PROGRAM SerialCom
VAR
	fbSerialControl : SerialLineControlADS;
	fbSendString	: SendString;
	fbReceiveString	: ReceiveString;
	
	bBarcodeReceivedReset_FE: F_TRIG;
END_VAR

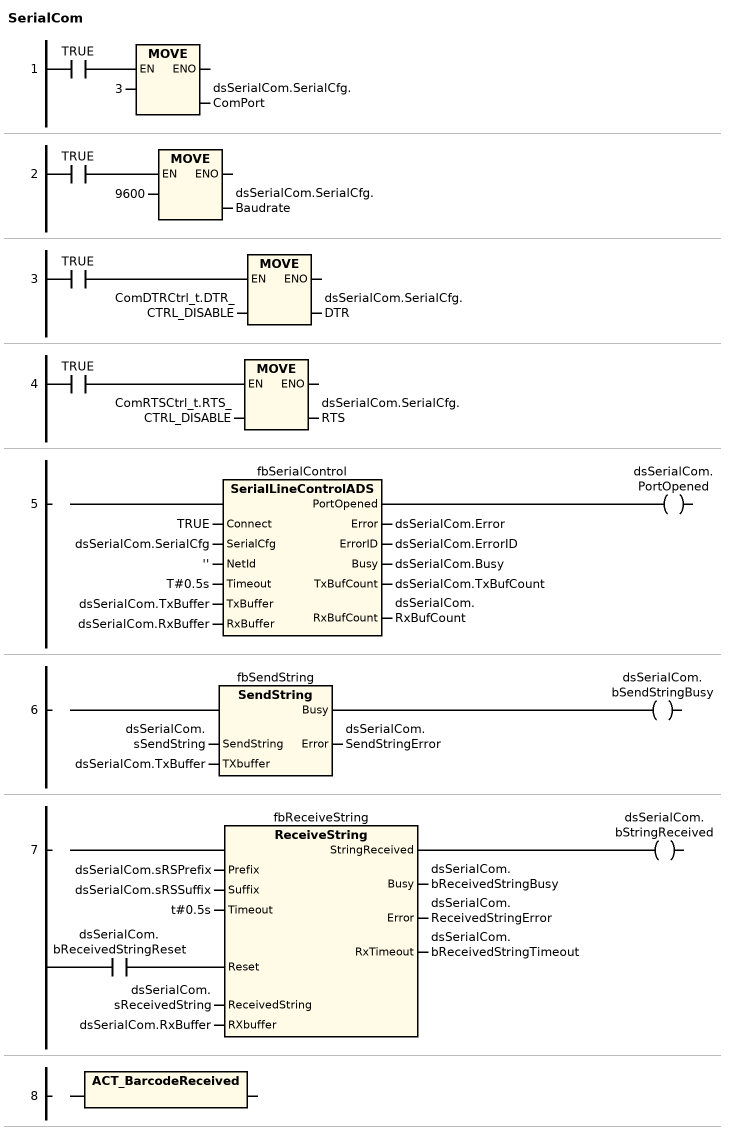
// NETWORK 1
dsSerialCom.SerialCfg.ComPort := 3;

// NETWORK 2
dsSerialCom.SerialCfg.Baudrate := 9600;

// NETWORK 3
dsSerialCom.SerialCfg.DTR := ComDTRCtrl_t.DTR_CTRL_DISABLE;

// NETWORK 4
dsSerialCom.SerialCfg.RTS := ComRTSCtrl_t.RTS_CTRL_DISABLE;

// NETWORK 5
fbSerialControl(
    Connect := TRUE,
    SerialCfg := dsSerialCom.SerialCfg,
    NetId := '',
    Timeout := T#0.5s,
    TxBuffer := dsSerialCom.TxBuffer,
    RxBuffer := dsSerialCom.RxBuffer,
    Error => dsSerialCom.Error,
    ErrorID => dsSerialCom.ErrorID,
    Busy => dsSerialCom.Busy,
    TxBufCount => dsSerialCom.TxBufCount,
    RxBufCount => dsSerialCom.RxBufCount); // SerialLineControlADS
dsSerialCom.PortOpened := fbSerialControl.PortOpened;

// NETWORK 6
fbSendString(
    SendString := dsSerialCom.sSendString,
    TXbuffer := dsSerialCom.TxBuffer,
    Error => dsSerialCom.SendStringError); // SendString
dsSerialCom.bSendStringBusy := fbSendString.Busy;

// NETWORK 7
fbReceiveString(
    Prefix := dsSerialCom.sRSPrefix,
    Suffix := dsSerialCom.sRSSuffix,
    Timeout := t#0.5s,
    Reset := dsSerialCom.bReceivedStringReset,
    ReceivedString := dsSerialCom.sReceivedString,
    RXbuffer := dsSerialCom.RxBuffer,
    Busy => dsSerialCom.bReceivedStringBusy,
    Error => dsSerialCom.ReceivedStringError,
    RxTimeout => dsSerialCom.bReceivedStringTimeout); // ReceiveString
dsSerialCom.bStringReceived := fbReceiveString.StringReceived;

// NETWORK 8
ACT_BarcodeReceived();

ACTION ACT_BarcodeReceived:

bBarcodeReceivedReset_FE(CLK:=((bAutoStartPb AND ARbDI[eX14000_LoadingConveyorSensor_Feed]) OR bBarcodeRegPage), Q=> );

IF bBarcodeReceivedReset_FE.Q THEN
dsSerialCom.sReceivedString:='';
END_IF
END_ACTION

END_PROGRAM

(* stored: Version 1.1.0.1, ProductVersion 3.1.4024.12
   POU SerialCom: Id {9be08231-d0f7-4c10-8f73-c2c448510bec}, SpecialFunc None
   Action ACT_BarcodeReceived: Id {4d8a6311-89a5-4813-b482-904c19279a94} *)
